Staubli VAL3: onFunctionEdit.pgx

public program onFunctionEdit(num x_nIndex, string x_sEvent, num x_nFunctionKey)
  local string l_sMessage
  local string l_sButton[2]
  local bool l_bOk
  local string l_sPage
  local string l_sItem
  local tool l_tTool
  local point l_pAlign
  local bool l_bYes
  local string l_sMessage2
begin
  //
  // do on Key action
  //
  // x_nIndex = actual index item
  // x_sEvent = actual event item
  //
  switch x_nFunctionKey
    // F1 button
    case 271
      // HERE POINT
      if !cycleStatus:bCycle
        call language:message(l_sMessage,160)
        call language:getYesNo(l_sButton)
        call use:yes_no(l_sMessage,l_sButton,l_bOk)
        if l_bOk
          call HerePoint(x_nIndex)
        endIf
      endIf
    break
    // F2 button
    case 272
      // ALIGN
      if !cycleStatus:bCycle
        resetMotion()
        call getFrame(fSetFrame,false)
        // tool
        call tcp:getTool(l_tTool,pEditPoint.nIndexTool)
        l_pAlign=here(l_tTool,world)
        l_pAlign.trsf=align(l_pAlign.trsf,fSetFrame.trsf)
        call language:message(l_sMessage,203)
        call language:message(l_sMessage2,134)
        l_sMessage=l_sMessage+" "+l_sMessage2+"..."
        call use:timerDialog(l_sMessage,0)
        movej(l_pAlign,l_tTool,mMdesc)
        watch(isEmpty() or isKeyPressed(255),3)
        if !isEmpty()
          resetMotion()
        endIf
        delay(2)
      endIf
    break
    // F3 button
    case 273
      // Select the gun
      l_sPage="Disk://kernel/page/tool"
      call loadPage(l_sPage,l_sItem)
      // set the tool
      pEditPoint.nIndexTool=saveData:nIndexTool
    break
    // F4 button
    case 274
    break
    // F5 button
    case 275
    break
    // F6 button
    case 276
      // change all the approach speed
      call changeSpeed(0,x_nIndex)
    break
    // F7 button
    case 277
      // change all the depart speed
      call changeSpeed(1,x_nIndex)
    break
    // F8 button
    case 278
      // save it
      bToSave=true
    break
  endSwitch
end
